// TIA Portal V19 export
DATA_BLOCK "CarriageLubr_Control"   // DB142
// stored: InstanceOfName Lubr_Valve, InstanceOfType FB
"Lubr_Valve"
   // VAR_INPUT
   //    AreaInterface : "AreaInterface";
   //    DataIn : Struct
   //       PbStartLubr : Bool;
   //       PbStopLubr : Bool;
   //       CycleFbk : Bool;
   //       ConnectorPlugged : Bool;
   //    END_STRUCT;
   //    CIn : Struct
   //       LubrEnable : Bool;
   //       ActualPosition : LReal;
   //       OperationDone : Bool;
   //    END_STRUCT;
   //    Config : "LubrValve_Config";
   //    Simulation : Bool;
   // END_VAR
   // VAR_OUTPUT
   //    MachineInterface : "MachineInterface";
   //    COut : Struct
   //       LubrReq : Bool;
   //    END_STRUCT;
   //    ValveCmd : Bool;
   // END_VAR
   // VAR_IN_OUT
   //    LubrInterface : "LubrValve_ITF";
   //    Pers : "LubrValve_Pers";
   // END_VAR
   // VAR
   //    Ctrl : Struct
   //       ManualReq : Bool;
   //       AutomaticReq : Bool;
   //       LubrReq : Bool;
   //       ValveCmd : Bool;
   //    END_STRUCT;
   //    Sts : Struct
   //       EstopDelayed : Bool;
   //       ValveEnabled : Bool;
   //       WorkEnable : Bool;
   //       CycleDone : Bool;
   //       LastFeed { ExternalAccessible := 'False'; ExternalVisible := 'False'; ExternalWritable := 'False'} : LReal;
   //       IsStandstill : Bool;
   //       AlarmsPresence : Bool;
   //       WarningsPresence : Bool;
   //    END_STRUCT;
   //    Alarm : "LubrValve_Alr";
   //    Warning : "LubrValve_Wng";
   //    HMI : "LubrValve_HMI";
   //    tonEStopDelayed : IEC_TIMER;
   //    tonCycleDoneON : IEC_TIMER;
   //    tonCycleDoneOFF : IEC_TIMER;
   //    tonManualCycleReset : IEC_TIMER;
   //    tonValveOn : IEC_TIMER;
   //    tonValveOff : IEC_TIMER;
   //    tonWorkTime : "TonEna";
   //    Aux_PbStartLubr : Bool;
   //    Pe_PbStartLubr : Bool;
   //    Aux_CyckeFkb : Bool;
   //    Pe_CycleFbk : Bool;
   //    Aux_OpDone : Bool;
   //    Pe_OpDone : Bool;
   //    Aux_ValveCount : Bool;
   //    Pe_ValveCount : Bool;
   // END_VAR
BEGIN
END_DATA_BLOCK
